// TIA Portal V19 export
TYPE "LEXCHANGETRAY_typeRollerIoSignalProcessValues_B2"
// simulated: Bool
// trayAutomaticFeedingDetectionU2Em6: Bool
// stored: Access Published
   STRUCT
      simulated : Bool;
      trayAutomaticFeedingDetectionU2Em6 : Bool;
   END_STRUCT;
END_TYPE
